KUKA KRL data list: ho_60101.dat

&ACCESS RVO2
&REL 599
&COMMENT Pega Lateral
&PARAM DISKPATH = KRC:\R1\Program\MANIPULACAO LTC
DEFDAT  ho_60101
;FOLD EXTERNAL DECLARATIONS;%{PE}%MKUKATPBASIS,%CEXT,%VCOMMON,%P
;FOLD GRIPPERTECH EXT
EXT  H50 (INT  :IN,INT  :IN,INT  :IN,GRP_TYP  :IN )
;ENDFOLD (GRIPPERTECH EXT)
;FOLD SPOTTECH EXT
EXT  USERSPOT (S_COMMAND  :IN,SPOT_TYPE  :IN )
;ENDFOLD (SPOTTECH EXT)
;FOLD BASISTECH EXT;%{PE}%MKUKATPBASIS,%CEXT,%VEXT,%P
EXT  BAS (BAS_COMMAND  :IN,REAL  :IN )
DECL INT SUCCESS
;ENDFOLD (BASISTECH EXT)
;FOLD USER EXT;%{E}%MKUKATPUSER,%CEXT,%VEXT,%P
;Make your modifications here

;ENDFOLD (USER EXT)
;ENDFOLD (EXTERNAL DECLARATIONS)

;# ============ START PATH : bh_p13060r1_ltc_01 =============
DECL FDAT FLHP040={TOOL_NO 2,BASE_NO 2,IPO_FRAME #BASE}
DECL E6POS XLHP040={X 838.254578,Y -5574.66309,Z -866.243774,A 89.6557083,B 0.696913004,C -102.786201,S 18,T 35,E1 0.0,E2 0.0,E3 0.0,E4 0.0,E5 0.0,E6 0.0}
DECL FDAT FLHP045={TOOL_NO 2,BASE_NO 2,IPO_FRAME #BASE}
DECL PDAT PP_OLP6={VEL 100.0,ACC 100.0,APO_DIST 100.0}
DECL E6POS XLHP045={X 1031.34094,Y -3395.22192,Z 766.315613,A 82.4350967,B -0.70792228,C -83.1183472,S 18,T 35,E1 0.0,E2 0.0,E3 0.0,E4 0.0,E5 0.0,E6 0.0}
DECL E6POS XLHP030={X 942.53479,Y -5582.48291,Z -837.87439,A 89.7051163,B 0.529519916,C -102.831596,S 2,T 35,E1 0.0,E2 0.0,E3 0.0,E4 0.0,E5 0.0,E6 0.0}
DECL FDAT FLHP030={TOOL_NO 2,BASE_NO 2,IPO_FRAME #BASE}
DECL PDAT PPDAT2={VEL 100.0,ACC 100.0,APO_DIST 5.0}
DECL PDAT PPDAT3={VEL 100.0,ACC 100.0,APO_DIST 100.0}
DECL GRP_SUGG_T LAST_GRP={NUMBER[] "1                       ",STATE[] "1                       ",PARAMS[] "GDAT7                   "}
DECL GRP_TYP GGDAT1={G_APO #NO,GRP_TIME 0.200000003,CTRL #OFF,DLY 0,DST 1}
DECL GRP_TYP GGDAT2={G_APO #NO,GRP_TIME 0.200000003,CTRL #OFF,DLY 0,DST 1}
DECL GRP_TYP GGDAT3={G_APO #NO,GRP_TIME 0.200000003,CTRL #OFF,DLY 0,DST 1}
DECL GRP_TYP GGDAT4={G_APO #NO,GRP_TIME 0.200000003,CTRL #OFF,DLY 0,DST 1}
DECL GRP_TYP GGDAT5={G_APO #NO,GRP_TIME 0.200000003,CTRL #OFF,DLY 0,DST 1}
DECL E6POS XLHP010={X -2658.55298,Y 1587.45496,Z 1512.15198,A -2.75169802,B 1.47639501,C -107.936096,S 18,T 35,E1 0.0,E2 0.0,E3 0.0,E4 0.0,E5 0.0,E6 0.0}
DECL FDAT FLHP010={TOOL_NO 2,BASE_NO 0,IPO_FRAME #BASE}
DECL E6POS XLHP015={X -2656.13208,Y 1744.65796,Z 1013.55701,A -2.75470901,B 1.48318195,C -108.002502,S 18,T 35,E1 0.0,E2 0.0,E3 0.0,E4 0.0,E5 0.0,E6 0.0}
DECL FDAT FLHP015={TOOL_NO 2,BASE_NO 0,IPO_FRAME #BASE}
DECL PDAT PPDAT17={VEL 100.0,ACC 100.0,APO_DIST 100.0}
DECL GRP_TYP GGDAT6={G_APO #NO,GRP_TIME 0.200000003,CTRL #OFF,DLY 0,DST 1}
DECL GRP_TYP GGDAT7={G_APO #NO,GRP_TIME 0.200000003,CTRL #OFF,DLY 0,DST 1}
DECL E6POS XLHP035={X 670.721191,Y -5574.84619,Z -901.981323,A 89.6396027,B 0.701093078,C -103.174599,S 18,T 35,E1 0.0,E2 0.0,E3 0.0,E4 0.0,E5 0.0,E6 0.0}
DECL FDAT FLHP035={TOOL_NO 2,BASE_NO 2,IPO_FRAME #BASE}
DECL PDAT PPDAT22={VEL 100.0,ACC 100.0,APO_DIST 5.0}
DECL PDAT PPDAT23={VEL 50.0,ACC 100.0,APO_DIST 10.0}
DECL E6POS XLHP075={X 1017.82898,Y -3148.71802,Z 1493.39404,A 4.49403811,B 78.8011627,C -170.569595,S 2,T 35,E1 0.0,E2 0.0,E3 0.0,E4 0.0,E5 0.0,E6 0.0}
DECL FDAT FLHP075={TOOL_NO 2,BASE_NO 2,IPO_FRAME #BASE}
DECL PDAT PPDAT24={VEL 100.0,ACC 100.0,APO_DIST 10.0}
DECL LDAT LCPDAT1={VEL 2.0,ACC 100.0,APO_DIST 100.0,APO_FAC 50.0}
DECL E6POS XPick_pos={X 581.659302,Y -5576.59277,Z -920.624817,A 89.7079163,B 1.09576297,C -102.428299,S 18,T 35,E1 0.0,E2 0.0,E3 0.0,E4 0.0,E5 0.0,E6 0.0}
DECL FDAT FPick_pos={TOOL_NO 2,BASE_NO 2,IPO_FRAME #BASE}
DECL E6POS XLHP005={X 1017.82898,Y -3148.71704,Z 1493.39502,A 4.49398613,B 78.8012009,C -170.569595,S 2,T 35,E1 0.0,E2 0.0,E3 0.0,E4 0.0,E5 0.0,E6 0.0}
DECL FDAT FLHP005={TOOL_NO 2,BASE_NO 2,IPO_FRAME #BASE}
DECL BASIS_SUGG_T LAST_BASIS={POINT1[] "LHP048                  ",POINT2[] "LHP048                  ",CP_PARAMS[] "CPDAT4                  ",PTP_PARAMS[] "PDAT12                  ",CONT[] "C_DIS                   ",CP_VEL[] "1                       ",PTP_VEL[] "100                     ",SYNC_PARAMS[] "SYNCDAT                 ",SPL_NAME[] "S0                      "}
DECL E6POS XLHP006={X -368.39151,Y 1361.11304,Z 1659.71802,A -0.79789108,B -0.378875285,C -112.862396,S 18,T 11,E1 0.0,E2 0.0,E3 0.0,E4 0.0,E5 0.0,E6 0.0}
DECL FDAT FLHP006={TOOL_NO 2,BASE_NO 0,IPO_FRAME #BASE,POINT2[] " ",TQ_STATE FALSE}
DECL PDAT PPDAT1={VEL 100.0,ACC 100.0,APO_DIST 100.0,GEAR_JERK 50.0}
DECL LDAT LCPDAT2={VEL 2.0,ACC 50.0,APO_DIST 100.0,APO_FAC 50.0,AXIS_VEL 100.0,AXIS_ACC 100.0,ORI_TYP #VAR,CIRC_TYP #BASE,JERK_FAC 50.0,GEAR_JERK 50.0,EXAX_IGN 0}
DECL E6POS XLHP007={X -1393.56396,Y 1405.05505,Z 1695.875,A -1.87000704,B 0.636861086,C -110.161598,S 18,T 35,E1 0.0,E2 0.0,E3 0.0,E4 0.0,E5 0.0,E6 0.0}
DECL FDAT FLHP007={TOOL_NO 2,BASE_NO 0,IPO_FRAME #BASE,POINT2[] " ",TQ_STATE FALSE}
DECL LDAT LCPDAT3={VEL 2.0,ACC 50.0,APO_DIST 100.0,APO_FAC 50.0,AXIS_VEL 100.0,AXIS_ACC 100.0,ORI_TYP #VAR,CIRC_TYP #BASE,JERK_FAC 50.0,GEAR_JERK 50.0,EXAX_IGN 0}
DECL E6POS XLHP008={X -1661.89697,Y 1549.32605,Z 1559.50305,A -2.13267398,B 0.891956985,C -109.509102,S 18,T 35,E1 0.0,E2 0.0,E3 0.0,E4 0.0,E5 0.0,E6 0.0}
DECL FDAT FLHP008={TOOL_NO 2,BASE_NO 0,IPO_FRAME #BASE,POINT2[] " ",TQ_STATE FALSE}
DECL LDAT LCPDAT4={VEL 2.0,ACC 50.0,APO_DIST 100.0,APO_FAC 50.0,AXIS_VEL 100.0,AXIS_ACC 100.0,ORI_TYP #VAR,CIRC_TYP #BASE,JERK_FAC 50.0,GEAR_JERK 50.0,EXAX_IGN 0}
DECL E6POS XLHP041={X 842.897827,Y -5574.10889,Z -655.778625,A 89.3989334,B -13.9881802,C -99.0561829,S 18,T 35,E1 0.0,E2 0.0,E3 0.0,E4 0.0,E5 0.0,E6 0.0}
DECL FDAT FLHP041={TOOL_NO 2,BASE_NO 2,IPO_FRAME #BASE,POINT2[] " ",TQ_STATE FALSE}
DECL PDAT PPDAT4={VEL 100.0,ACC 100.0,APO_DIST 100.0,APO_MODE #CDIS,GEAR_JERK 50.0}
DECL E6POS XLHP042={X 906.871277,Y -5577.9292,Z 95.8650284,A 88.6567383,B -2.11703706,C -92.0317688,S 18,T 35,E1 0.0,E2 0.0,E3 0.0,E4 0.0,E5 0.0,E6 0.0}
DECL FDAT FLHP042={TOOL_NO 2,BASE_NO 2,IPO_FRAME #BASE,POINT2[] " ",TQ_STATE FALSE}
DECL PDAT PPDAT5={VEL 100.0,ACC 100.0,APO_DIST 100.0,APO_MODE #CDIS,GEAR_JERK 50.0}
DECL E6POS XLHP043={X 1144.5,Y -4762.86719,Z 491.821686,A 88.659668,B -2.11881399,C -92.0398865,S 18,T 35,E1 0.0,E2 0.0,E3 0.0,E4 0.0,E5 0.0,E6 0.0}
DECL FDAT FLHP043={TOOL_NO 2,BASE_NO 2,IPO_FRAME #BASE,POINT2[] " ",TQ_STATE FALSE}
DECL PDAT PPDAT6={VEL 100.0,ACC 100.0,APO_DIST 100.0,APO_MODE #CDIS,GEAR_JERK 50.0}
DECL E6POS XLHP044={X 1150.29895,Y -3570.01807,Z 487.99411,A 88.6528091,B -2.07348609,C -92.0989532,S 18,T 35,E1 0.0,E2 0.0,E3 0.0,E4 0.0,E5 0.0,E6 0.0}
DECL FDAT FLHP044={TOOL_NO 2,BASE_NO 2,IPO_FRAME #BASE,POINT2[] " ",TQ_STATE FALSE}
DECL PDAT PPDAT7={VEL 100.0,ACC 100.0,APO_DIST 100.0,APO_MODE #CDIS,GEAR_JERK 50.0}
DECL E6POS XLHP043A={X 1238.22302,Y -4533.76221,Z 526.550171,A 88.7746582,B -1.41036403,C -91.4281235,S 18,T 35,E1 0.0,E2 0.0,E3 0.0,E4 0.0,E5 0.0,E6 0.0}
DECL FDAT FLHP043a={TOOL_NO 2,BASE_NO 2,IPO_FRAME #BASE,POINT2[] " ",TQ_STATE FALSE}
DECL PDAT PPDAT8={VEL 100.0,ACC 100.0,APO_DIST 100.0,APO_MODE #CDIS,GEAR_JERK 50.0}
DECL E6POS XLHP046={X 1011.28198,Y -3329.18994,Z 1023.70502,A 78.8528366,B 27.6525898,C -87.816452,S 18,T 35,E1 0.0,E2 0.0,E3 0.0,E4 0.0,E5 0.0,E6 0.0}
DECL FDAT FLHP046={TOOL_NO 2,BASE_NO 2,IPO_FRAME #BASE,POINT2[] " ",TQ_STATE FALSE}
DECL PDAT PPDAT9={VEL 100.0,ACC 100.0,APO_DIST 100.0,APO_MODE #CDIS,GEAR_JERK 50.0}
DECL PDAT PPDAT11={VEL 100.0,ACC 100.0,APO_DIST 15.0,APO_MODE #CDIS,GEAR_JERK 50.0}
DECL E6POS XLHP048={X -1185.21997,Y 1414.68799,Z 1799.43298,A -2.28385901,B -1.065395,C -115.208,S 18,T 35,E1 0.0,E2 0.0,E3 0.0,E4 0.0,E5 0.0,E6 0.0}
DECL FDAT FLHP048={TOOL_NO 2,BASE_NO 0,IPO_FRAME #BASE,POINT2[] " ",TQ_STATE FALSE}
DECL PDAT PPDAT12={VEL 100.0,ACC 100.0,APO_DIST 15.0,APO_MODE #CDIS,GEAR_JERK 50.0}
DECL PDAT PPDAT13={VEL 100.0,ACC 100.0,APO_DIST 15.0,APO_MODE #CDIS,GEAR_JERK 50.0}
DECL PDAT PPDAT14={VEL 100.0,ACC 100.0,APO_DIST 15.0,APO_MODE #CDIS,GEAR_JERK 50.0}
ENDDAT
